TYPE ST_AuxiliaryPowerValues :
	STRUCT
		index:USINT;		//Indice
		channel:USINT;		//Canal
		value:DINT;			//Valor
	END_STRUCT
END_TYPE

(* stored: Version 1.1.0.1, ProductVersion 3.1.4024.12
   DUT ST_AuxiliaryPowerValues: Id {2966667f-42f9-4743-83ad-a241daca0602} *)
